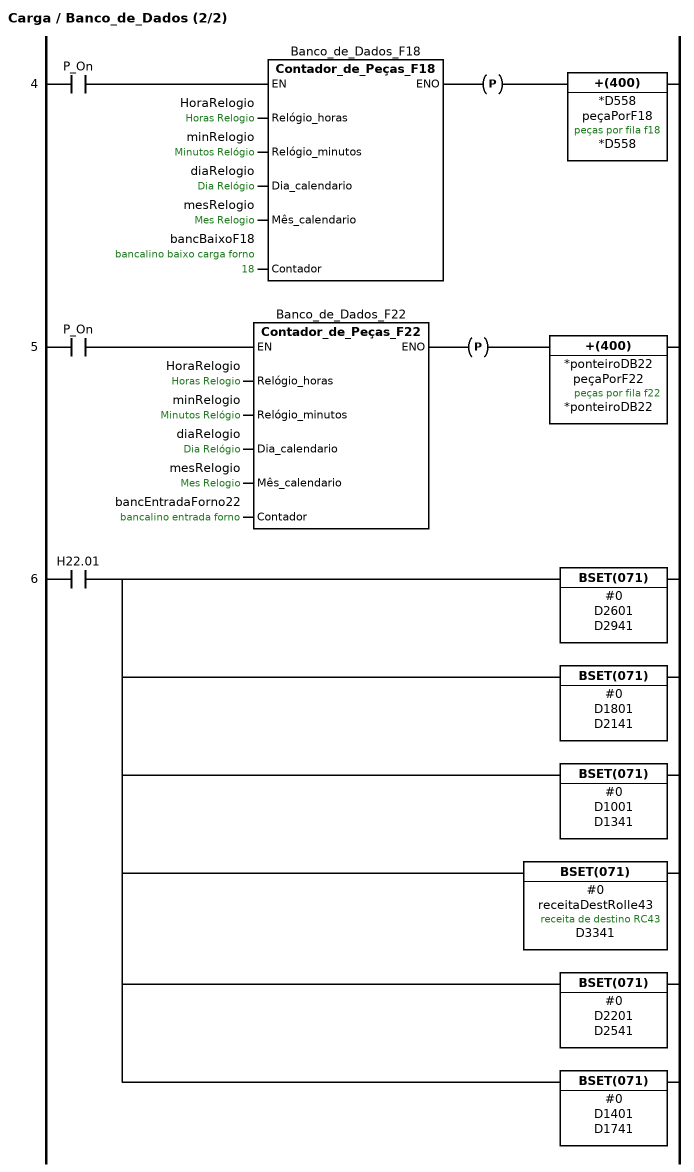
; [picture p24: Carga / Banco_de_Dados, rungs 4-6]
; rung 4
LD P_On
CALL Banco_de_Dados_F18 : Contador_de_Peças_F18 (Relógio_horas := HoraRelogio, Relógio_minutos := minRelogio, Dia_calendario := diaRelogio, Mês_calendario := mesRelogio, Contador := bancBaixoF18)  ; Horas Relogio, Minutos Relógio, Dia Relógio, Mes Relogio, bancalino baixo carga forno 18
UP(521)
+(400) *D558 peçaPorF18 *D558  ; peças por fila f18
; rung 5
LD P_On
CALL Banco_de_Dados_F22 : Contador_de_Peças_F22 (Relógio_horas := HoraRelogio, Relógio_minutos := minRelogio, Dia_calendario := diaRelogio, Mês_calendario := mesRelogio, Contador := bancEntradaForno22)  ; Horas Relogio, Minutos Relógio, Dia Relógio, Mes Relogio, bancalino entrada forno
UP(521)
+(400) *ponteiroDB22 peçaPorF22 *ponteiroDB22  ; peças por fila f22
; rung 6
LD H22.01
BSET(071) #0 D2601 D2941
BSET(071) #0 D1801 D2141
BSET(071) #0 D1001 D1341
BSET(071) #0 receitaDestRolle43 D3341  ; receita de destino RC43
BSET(071) #0 D2201 D2541
BSET(071) #0 D1401 D1741

### Section Transferencia_excel

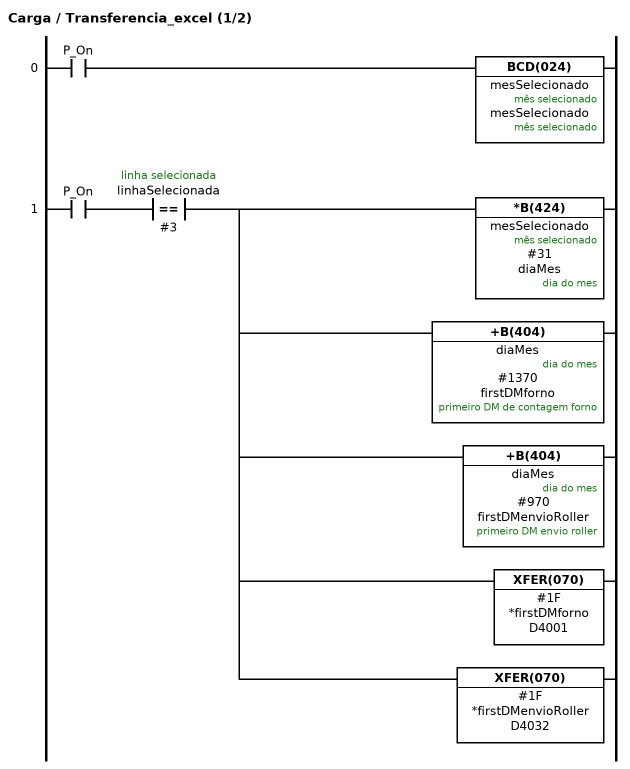
; rung 0
LD P_On
BCD(024) mesSelecionado mesSelecionado  ; mês selecionado
; rung 1
LD P_On
AND=(300) linhaSelecionada #3  ; linha selecionada
*B(424) mesSelecionado #31 diaMes  ; mês selecionado, dia do mes
+B(404) diaMes #1370 firstDMforno  ; dia do mes, primeiro DM de contagem forno
+B(404) diaMes #970 firstDMenvioRoller  ; dia do mes, primeiro DM envio roller
XFER(070) #1F *firstDMforno D4001
XFER(070) #1F *firstDMenvioRoller D4032

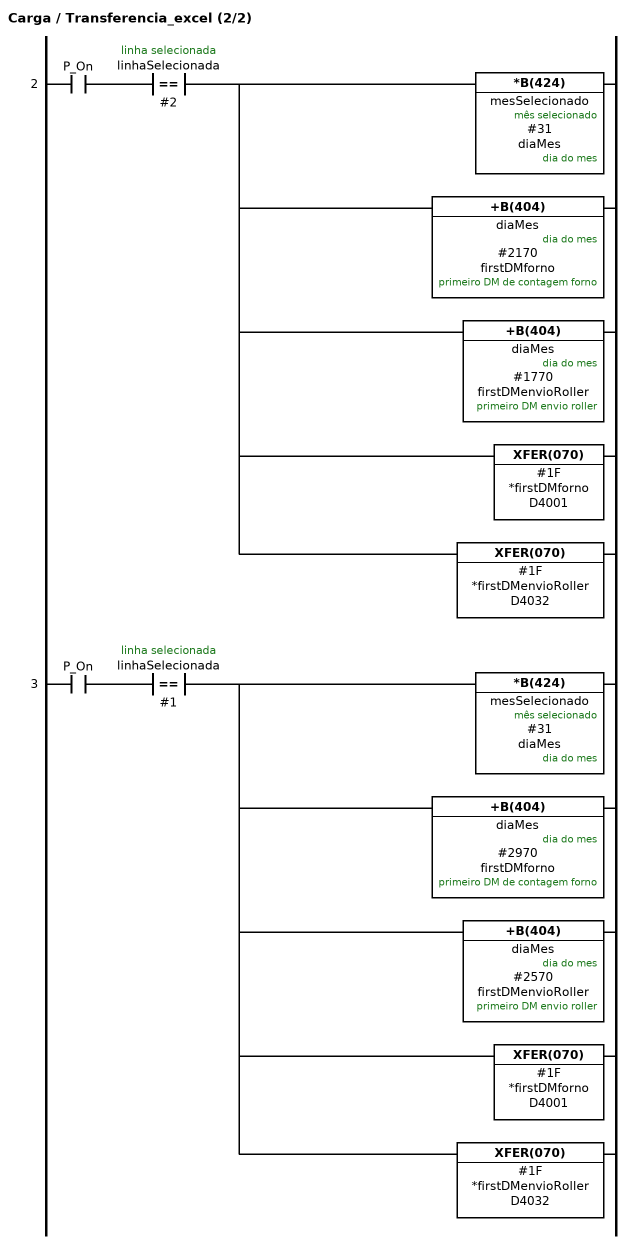
; rung 2
LD P_On
AND=(300) linhaSelecionada #2  ; linha selecionada
*B(424) mesSelecionado #31 diaMes  ; mês selecionado, dia do mes
+B(404) diaMes #2170 firstDMforno  ; dia do mes, primeiro DM de contagem forno
+B(404) diaMes #1770 firstDMenvioRoller  ; dia do mes, primeiro DM envio roller
XFER(070) #1F *firstDMforno D4001
XFER(070) #1F *firstDMenvioRoller D4032
; rung 3
LD P_On
AND=(300) linhaSelecionada #1  ; linha selecionada
*B(424) mesSelecionado #31 diaMes  ; mês selecionado, dia do mes
+B(404) diaMes #2970 firstDMforno  ; dia do mes, primeiro DM de contagem forno
+B(404) diaMes #2570 firstDMenvioRoller  ; dia do mes, primeiro DM envio roller
XFER(070) #1F *firstDMforno D4001
XFER(070) #1F *firstDMenvioRoller D4032

### Section Relogio

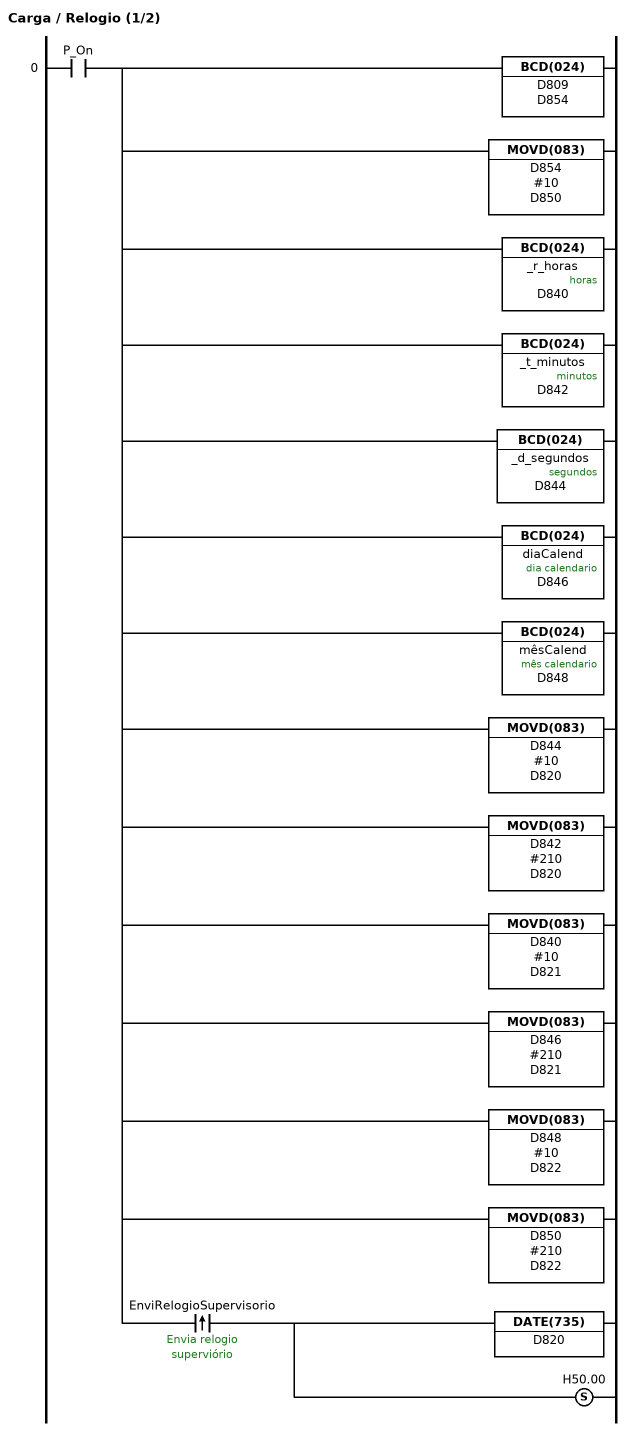
; rung 0
LD P_On
BCD(024) D809 D854
MOVD(083) D854 #10 D850
BCD(024) _r_horas D840  ; horas
BCD(024) _t_minutos D842  ; minutos
BCD(024) _d_segundos D844  ; segundos
BCD(024) diaCalend D846  ; dia calendario
BCD(024) mêsCalend D848  ; mês calendario
MOVD(083) D844 #10 D820
MOVD(083) D842 #210 D820
MOVD(083) D840 #10 D821
MOVD(083) D846 #210 D821
MOVD(083) D848 #10 D822
MOVD(083) D850 #210 D822
@AND EnviRelogioSupervisorio  ; Envia relogio superviório
DATE(735) D820
SET H50.00

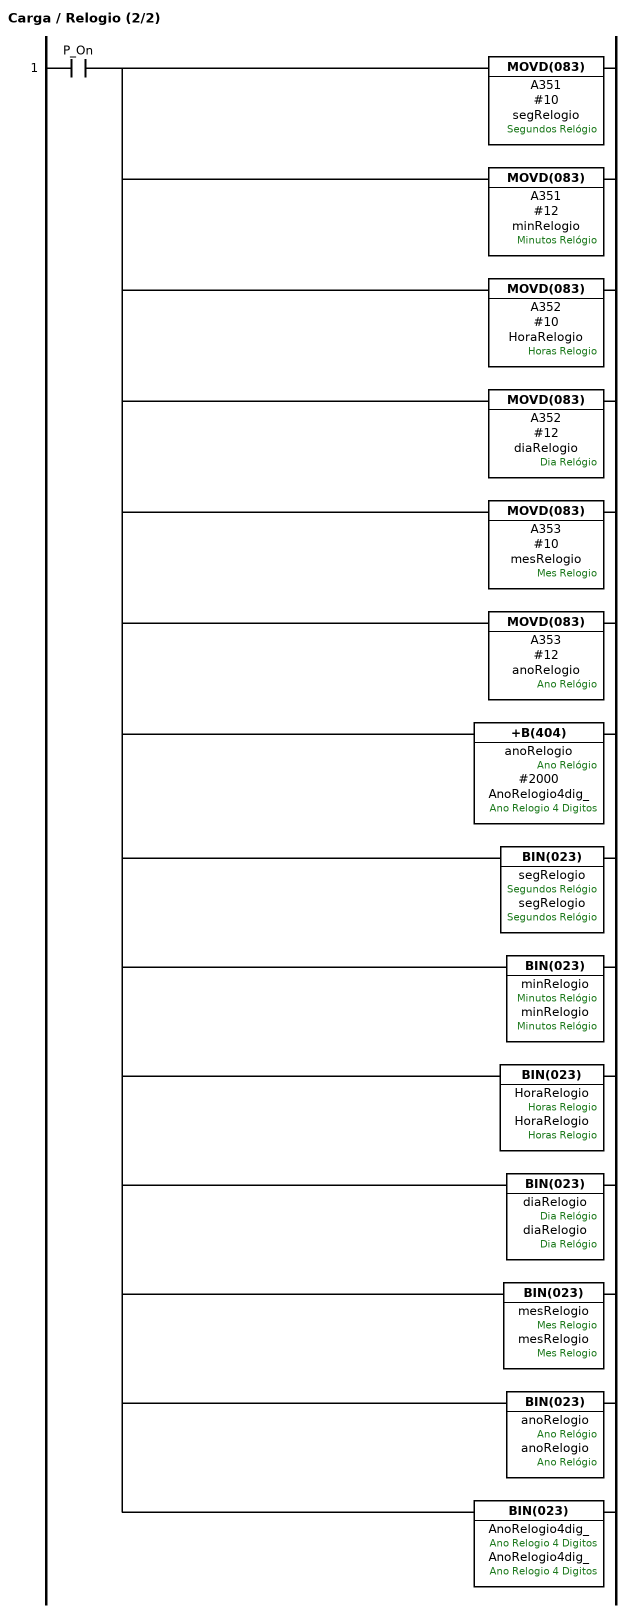
; rung 1
LD P_On
MOVD(083) A351 #10 segRelogio  ; Segundos Relógio
MOVD(083) A351 #12 minRelogio  ; Minutos Relógio
MOVD(083) A352 #10 HoraRelogio  ; Horas Relogio
MOVD(083) A352 #12 diaRelogio  ; Dia Relógio
MOVD(083) A353 #10 mesRelogio  ; Mes Relogio
MOVD(083) A353 #12 anoRelogio  ; Ano Relógio
+B(404) anoRelogio #2000 AnoRelogio4dig_  ; Ano Relógio, Ano Relogio 4 Digitos
BIN(023) segRelogio segRelogio  ; Segundos Relógio
BIN(023) minRelogio minRelogio  ; Minutos Relógio
BIN(023) HoraRelogio HoraRelogio  ; Horas Relogio
BIN(023) diaRelogio diaRelogio  ; Dia Relógio
BIN(023) mesRelogio mesRelogio  ; Mes Relogio
BIN(023) anoRelogio anoRelogio  ; Ano Relógio
BIN(023) AnoRelogio4dig_ AnoRelogio4dig_  ; Ano Relogio 4 Digitos

### Section End
; rung 0
END(001)

## Program Escolha41 (cyclic task 2)
Local symbols
TIM 4.12 BOOL
anoRelogio D328 CHANNEL  ; Ano relógio
bit2 BOOL
box1 4.01 BOOL  ; box1
box2 4.02 BOOL  ; box2
box3 4.03 BOOL  ; box3
box4 4.04 BOOL  ; box4
box5 4.05 BOOL  ; box5
box6 4.06 BOOL  ; box6
caco 4.00 BOOL  ; caco
cntAmostragem D316 CHANNEL  ; contador amostragem
cntBox0 D300 CHANNEL  ; contagem box 0
cntBox1 D302 CHANNEL  ; contagem box 1
cntBox2 D304 CHANNEL  ; contagem box 2
cntBox3 D306 CHANNEL  ; contagem box 3
cntBox4 D308 CHANNEL  ; contagem box 4
cntBox5 D310 CHANNEL  ; contagem box 5
cntBox6 D312 CHANNEL  ; contagem box 6
cntTotal D314 CHANNEL  ; contagem total
d400D400 CHANNEL
diaRelogio D324 CHANNEL  ; Dia relógio
enviaRelogio H12.00 BOOL  ; envia relogio
horEnvio D336 CHANNEL  ; hora de envio
horIHM D330 CHANNEL  ; hora ihm
horRelogio D322 CHANNEL  ; Horas relógio
mesRelogio D326 CHANNEL  ; Mes Relógio
minIHM D332 CHANNEL  ; minuto ihm
minRelogio D320 CHANNEL  ; Minutos relógio
mitEnvio D338 CHANNEL  ; minuto envio
resetCnt 4.07 BOOL  ; reset contagem
segEnvio D340 CHANNEL  ; segundo envio
segIHM D334 CHANNEL  ; segundo ihm
segRelogio D318 CHANNEL  ; Segundos Relógio
selecaoCom 4.09 BOOL  ; seleção comercial
totalPc 4.08 BOOL  ; total peças

### Section Controle_Qualidade

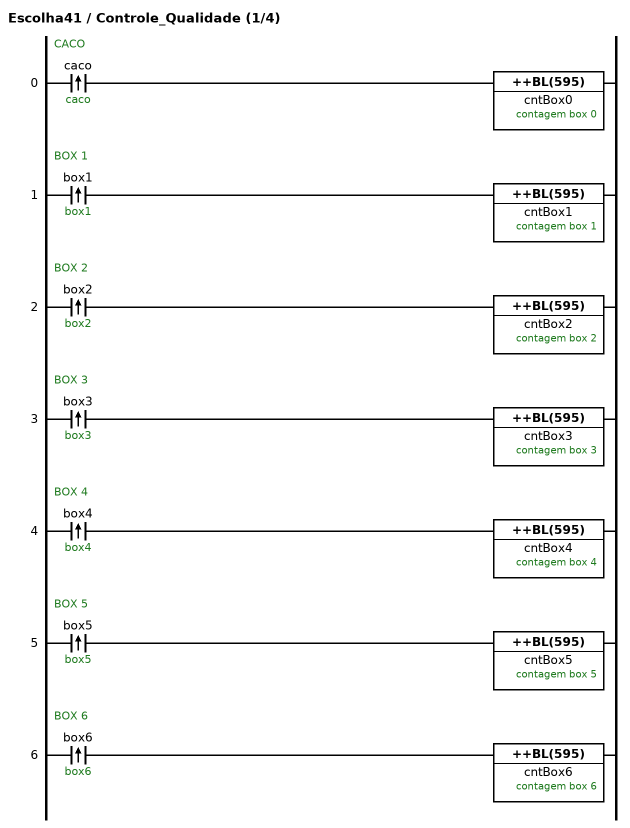
; rung 0: CACO
@LD caco  ; caco
++BL(595) cntBox0  ; contagem box 0
; rung 1: BOX 1
@LD box1  ; box1
++BL(595) cntBox1  ; contagem box 1
; rung 2: BOX 2
@LD box2  ; box2
++BL(595) cntBox2  ; contagem box 2
; rung 3: BOX 3
@LD box3  ; box3
++BL(595) cntBox3  ; contagem box 3
; rung 4: BOX 4
@LD box4  ; box4
++BL(595) cntBox4  ; contagem box 4
; rung 5: BOX 5
@LD box5  ; box5
++BL(595) cntBox5  ; contagem box 5
; rung 6: BOX 6
@LD box6  ; box6
++BL(595) cntBox6  ; contagem box 6

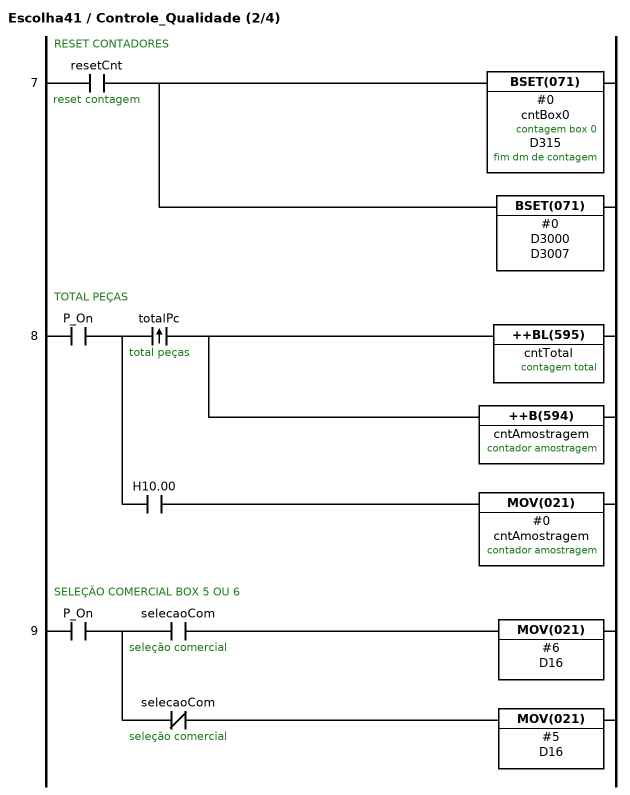
; rung 7: RESET CONTADORES
LD resetCnt  ; reset contagem
BSET(071) #0 cntBox0 D315  ; contagem box 0, fim dm de contagem
BSET(071) #0 D3000 D3007
; rung 8: TOTAL PEÇAS
LD P_On
OUT TR0
@AND totalPc  ; total peças
++BL(595) cntTotal  ; contagem total
++B(594) cntAmostragem  ; contador amostragem
LD TR0
AND H10.00
MOV(021) #0 cntAmostragem  ; contador amostragem
; rung 9: SELEÇÃO COMERCIAL BOX 5 OU 6
LD P_On
OUT TR0
AND selecaoCom  ; seleção comercial
MOV(021) #6 D16
LD TR0
ANDNOT selecaoCom  ; seleção comercial
MOV(021) #5 D16

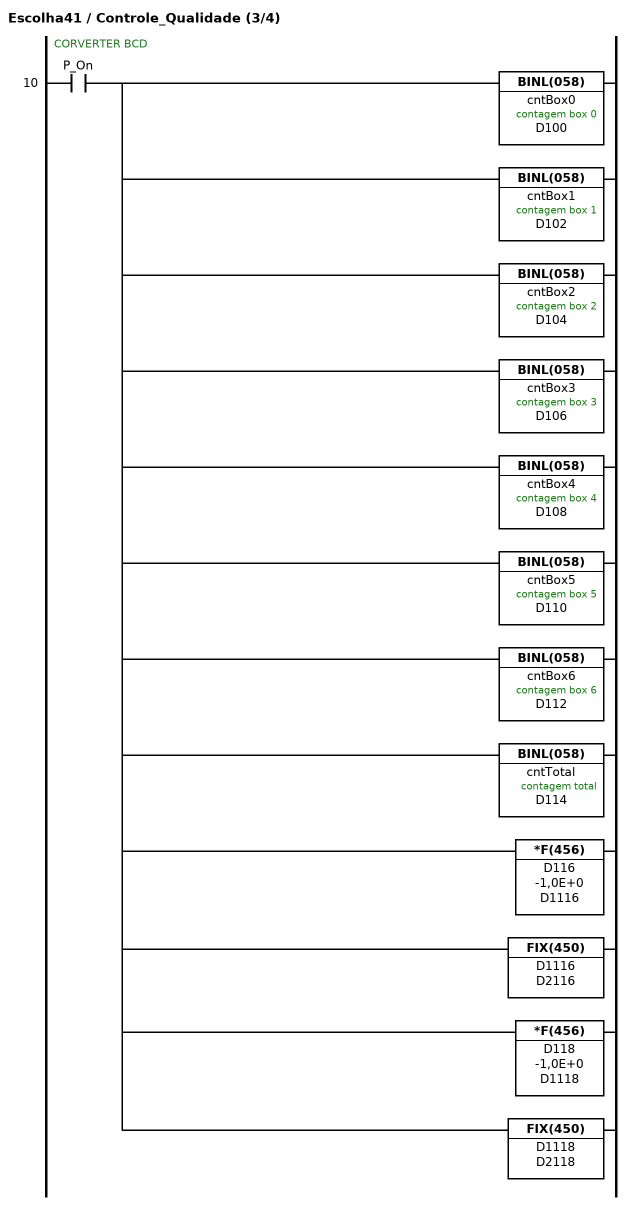
; rung 10: CORVERTER BCD
LD P_On
BINL(058) cntBox0 D100  ; contagem box 0
BINL(058) cntBox1 D102  ; contagem box 1
BINL(058) cntBox2 D104  ; contagem box 2
BINL(058) cntBox3 D106  ; contagem box 3
BINL(058) cntBox4 D108  ; contagem box 4
BINL(058) cntBox5 D110  ; contagem box 5
BINL(058) cntBox6 D112  ; contagem box 6
BINL(058) cntTotal D114  ; contagem total
*F(456) D116 -1,0E+0 D1116
FIX(450) D1116 D2116
*F(456) D118 -1,0E+0 D1118
FIX(450) D1118 D2118

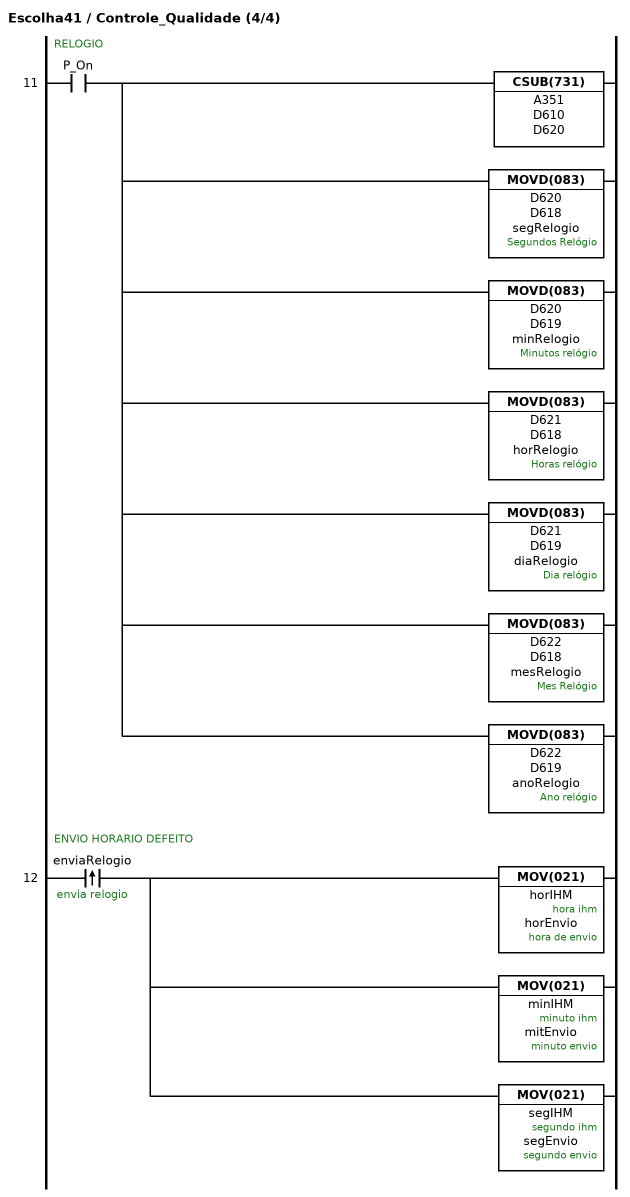
; rung 11: RELOGIO
LD P_On
CSUB(731) A351 D610 D620
MOVD(083) D620 D618 segRelogio  ; Segundos Relógio
MOVD(083) D620 D619 minRelogio  ; Minutos relógio
MOVD(083) D621 D618 horRelogio  ; Horas relógio
MOVD(083) D621 D619 diaRelogio  ; Dia relógio
MOVD(083) D622 D618 mesRelogio  ; Mes Relógio
MOVD(083) D622 D619 anoRelogio  ; Ano relógio
; rung 12: ENVIO HORARIO DEFEITO
@LD enviaRelogio  ; envia relogio
MOV(021) horIHM horEnvio  ; hora ihm, hora de envio
MOV(021) minIHM mitEnvio  ; minuto ihm, minuto envio
MOV(021) segIHM segEnvio  ; segundo ihm, segundo envio

### Section END
; rung 0
END(001)

## Program Escolha43 (cyclic task 3)
Local symbols
TIM 5.12 BOOL
anoRelogio D428 CHANNEL  ; Ano relógio
bit2 BOOL
box1 5.01 BOOL  ; box1
box2 5.02 BOOL  ; box2
box3 5.03 BOOL  ; box3
box4 5.04 BOOL  ; box4
box5 5.05 BOOL  ; box5
box6 5.06 BOOL  ; box6
caco 5.00 BOOL  ; caco
cntAmostragem D416 CHANNEL  ; contador amostragem
cntBox0 D400 CHANNEL  ; contagem box 0
cntBox1 D402 CHANNEL  ; contagem box 1
cntBox2 D404 CHANNEL  ; contagem box 2
cntBox3 D406 CHANNEL  ; contagem box 3
cntBox4 D408 CHANNEL  ; contagem box 4
cntBox5 D410 CHANNEL  ; contagem box 5
cntBox6 D412 CHANNEL  ; contagem box 6
cntTotal D414 CHANNEL  ; contagem total
d400D400 CHANNEL
diaRelogio D424 CHANNEL  ; Dia relógio
enviaRelogio H13.01 BOOL  ; envia relogio
horEnvio D436 CHANNEL  ; hora de envio
horIHM D430 CHANNEL  ; hora ihm
horRelogio D422 CHANNEL  ; Horas relógio
mesRelogio D426 CHANNEL  ; Mes Relógio
minIHM D432 CHANNEL  ; minuto ihm
minRelogio D420 CHANNEL  ; Minutos relógio
mitEnvio D438 CHANNEL  ; minuto envio
resetCnt 5.07 BOOL  ; reset contagem
resetCntH H13.00 BOOL  ; reset contador
segEnvio D440 CHANNEL  ; segundo envio
segIHM D434 CHANNEL  ; segundo ihm
segRelogio D418 CHANNEL  ; Segundos Relógio
selecaoCom 5.09 BOOL  ; seleção comercial
totalPc 5.08 BOOL  ; total peças

### Section Controle_Qualidade

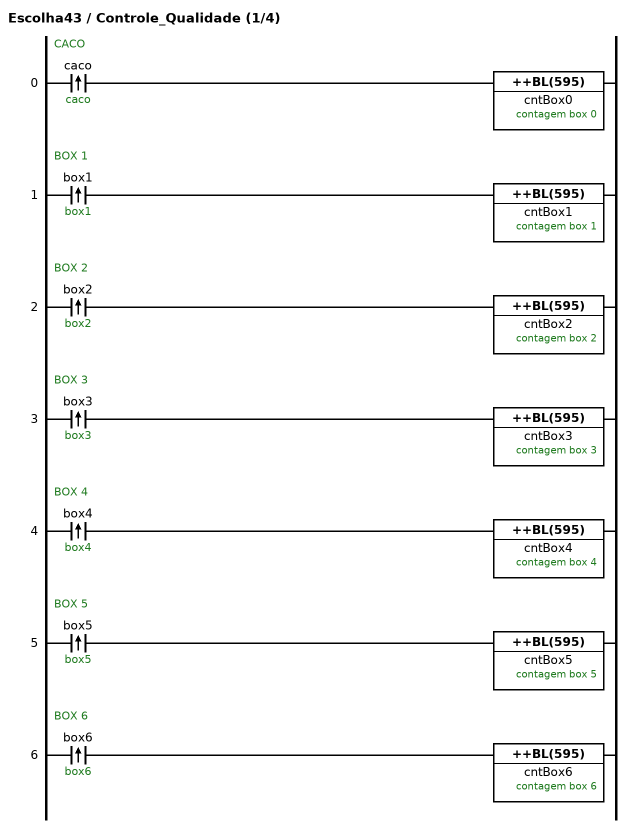
; rung 0: CACO
@LD caco  ; caco
++BL(595) cntBox0  ; contagem box 0
; rung 1: BOX 1
@LD box1  ; box1
++BL(595) cntBox1  ; contagem box 1
; rung 2: BOX 2
@LD box2  ; box2
++BL(595) cntBox2  ; contagem box 2
; rung 3: BOX 3
@LD box3  ; box3
++BL(595) cntBox3  ; contagem box 3
; rung 4: BOX 4
@LD box4  ; box4
++BL(595) cntBox4  ; contagem box 4
; rung 5: BOX 5
@LD box5  ; box5
++BL(595) cntBox5  ; contagem box 5
; rung 6: BOX 6
@LD box6  ; box6
++BL(595) cntBox6  ; contagem box 6

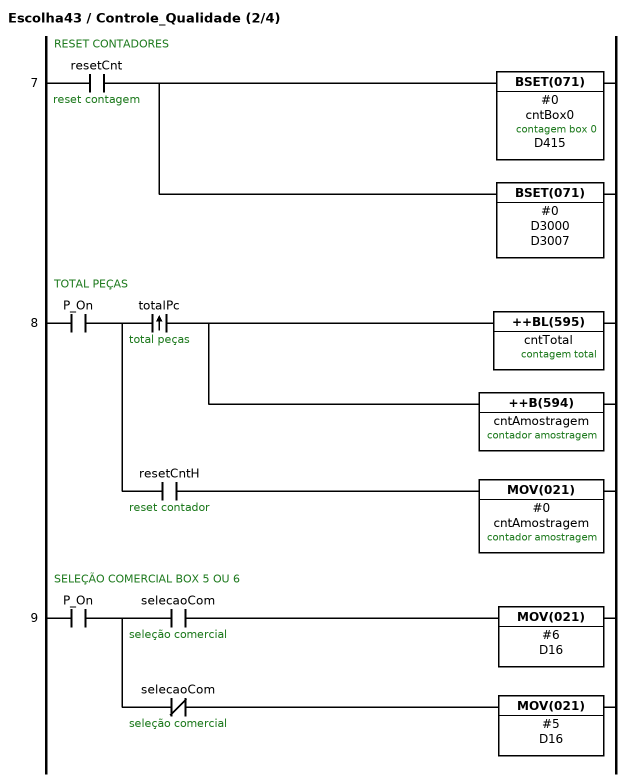
; rung 7: RESET CONTADORES
LD resetCnt  ; reset contagem
BSET(071) #0 cntBox0 D415  ; contagem box 0
BSET(071) #0 D3000 D3007
; rung 8: TOTAL PEÇAS
LD P_On
OUT TR0
@AND totalPc  ; total peças
++BL(595) cntTotal  ; contagem total
++B(594) cntAmostragem  ; contador amostragem
LD TR0
AND resetCntH  ; reset contador
MOV(021) #0 cntAmostragem  ; contador amostragem
; rung 9: SELEÇÃO COMERCIAL BOX 5 OU 6
LD P_On
OUT TR0
AND selecaoCom  ; seleção comercial
MOV(021) #6 D16
LD TR0
ANDNOT selecaoCom  ; seleção comercial
MOV(021) #5 D16

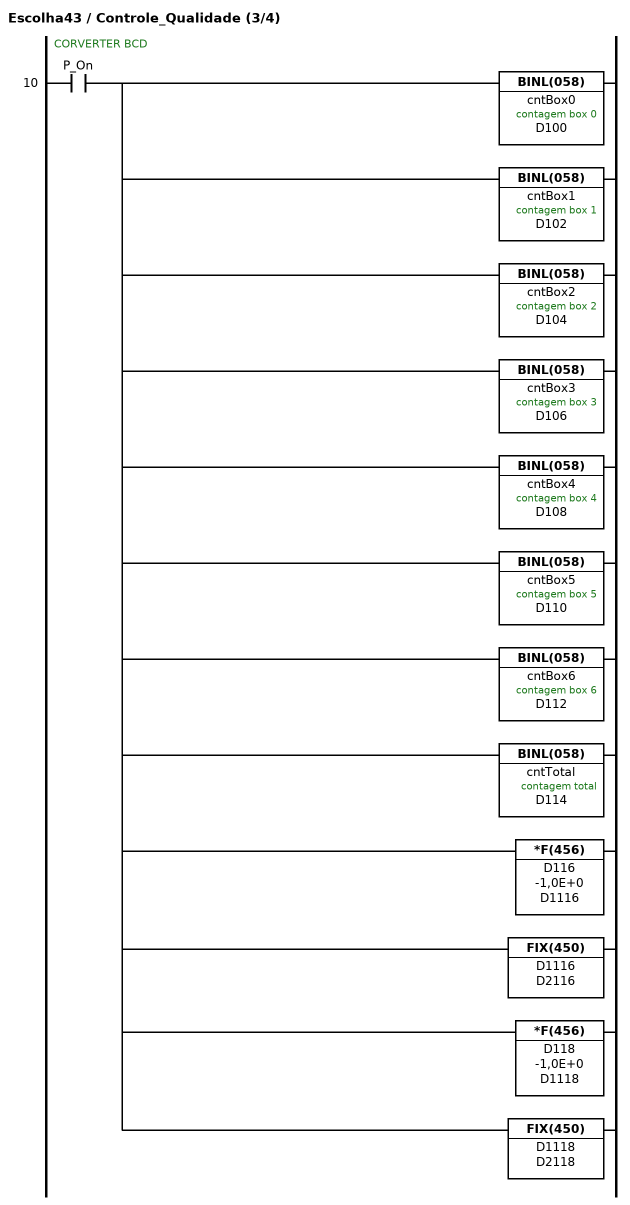
; rung 10: CORVERTER BCD
LD P_On
BINL(058) cntBox0 D100  ; contagem box 0
BINL(058) cntBox1 D102  ; contagem box 1
BINL(058) cntBox2 D104  ; contagem box 2
BINL(058) cntBox3 D106  ; contagem box 3
BINL(058) cntBox4 D108  ; contagem box 4
BINL(058) cntBox5 D110  ; contagem box 5
BINL(058) cntBox6 D112  ; contagem box 6
BINL(058) cntTotal D114  ; contagem total
*F(456) D116 -1,0E+0 D1116
FIX(450) D1116 D2116
*F(456) D118 -1,0E+0 D1118
FIX(450) D1118 D2118

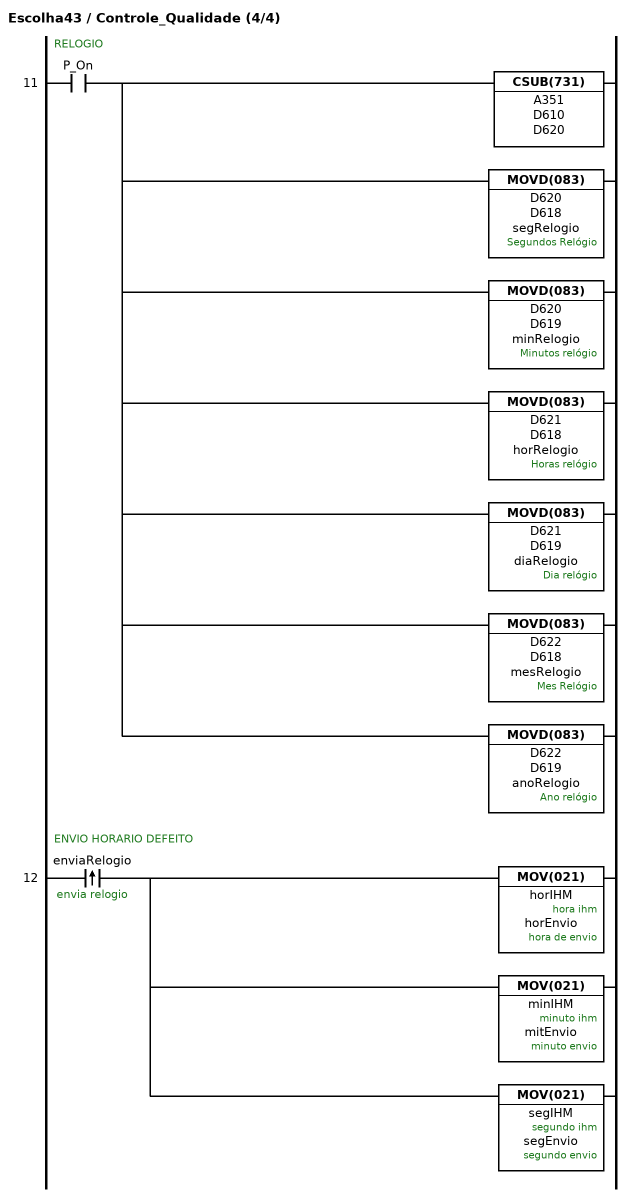
; rung 11: RELOGIO
LD P_On
CSUB(731) A351 D610 D620
MOVD(083) D620 D618 segRelogio  ; Segundos Relógio
MOVD(083) D620 D619 minRelogio  ; Minutos relógio
MOVD(083) D621 D618 horRelogio  ; Horas relógio
MOVD(083) D621 D619 diaRelogio  ; Dia relógio
MOVD(083) D622 D618 mesRelogio  ; Mes Relógio
MOVD(083) D622 D619 anoRelogio  ; Ano relógio
; rung 12: ENVIO HORARIO DEFEITO
@LD enviaRelogio  ; envia relogio
MOV(021) horIHM horEnvio  ; hora ihm, hora de envio
MOV(021) minIHM mitEnvio  ; minuto ihm, minuto envio
MOV(021) segIHM segEnvio  ; segundo ihm, segundo envio

### Section END
; rung 0
END(001)

## Function block Contador_de_Peças_F17
VAR_INPUT
  Relógio_horas : WORD;
  Relógio_minutos : WORD;
  Dia_calendario : WORD;
  Mês_calendario : WORD;
  Contador : BOOL;
END_VAR
VAR
  _31dias_vezes_2 AT D530 : WORD;
  Ponteiro_DWord AT D532 : WORD;
  Memória_de_Armazenagem AT D534 : WORD;
  Memoria_contagem_BIN AT D536 : WORD;
  Memoria_contagem_BCD AT D538 : WORD;
END_VAR

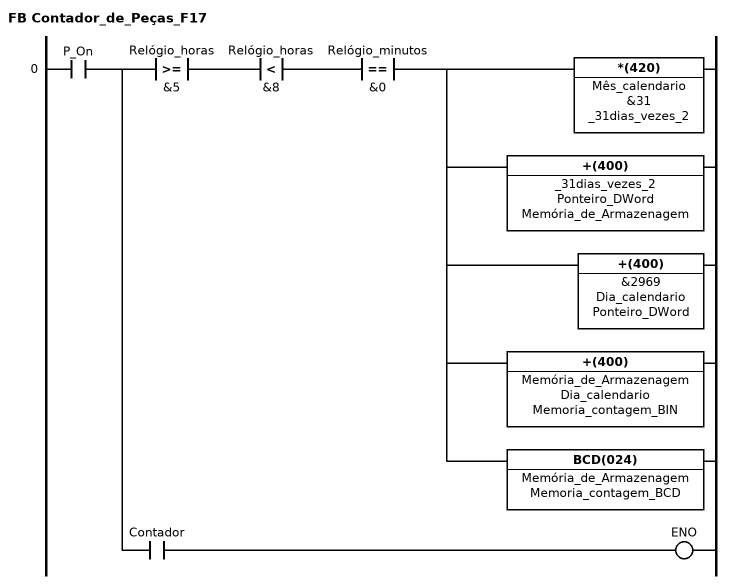
; rung 0
LD P_On
OUT TR0
AND>=(325) Relógio_horas &5
AND<(310) Relógio_horas &8
AND=(300) Relógio_minutos &0
*(420) Mês_calendario &31 _31dias_vezes_2
+(400) _31dias_vezes_2 Ponteiro_DWord Memória_de_Armazenagem
+(400) &2969 Dia_calendario Ponteiro_DWord
+(400) Memória_de_Armazenagem Dia_calendario Memoria_contagem_BIN
BCD(024) Memória_de_Armazenagem Memoria_contagem_BCD
LD TR0
AND Contador
OUT ENO

## Function block Contador_de_Peças_F18
VAR_INPUT
  Relógio_horas : WORD;
  Relógio_minutos : WORD;
  Dia_calendario : WORD;
  Mês_calendario : WORD;
  Contador : BOOL;
END_VAR
VAR
  _31dias_vezes_2 AT D550 : WORD;
  Ponteiro_DWord AT D552 : WORD;
  Memória_de_Armazenagem AT D554 : WORD;
  Memoria_contagem_BIN AT D556 : WORD;
  Memoria_contagem_BCD AT D558 : WORD;
END_VAR

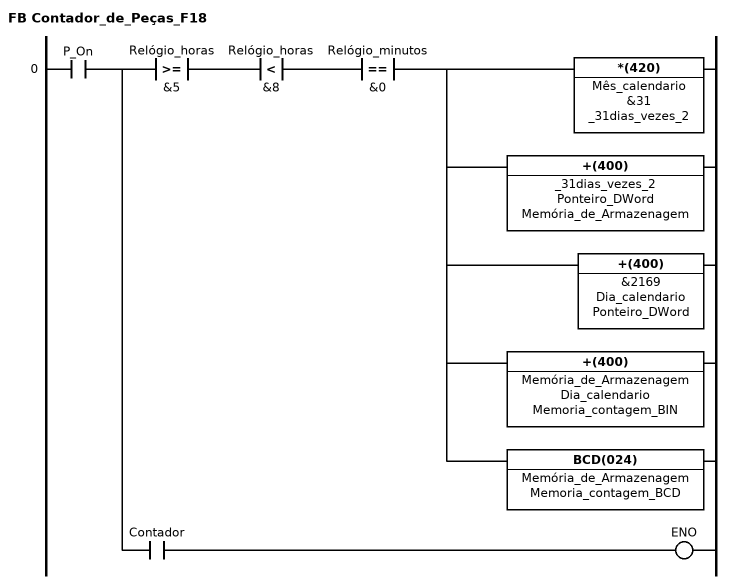
; rung 0
LD P_On
OUT TR0
AND>=(325) Relógio_horas &5
AND<(310) Relógio_horas &8
AND=(300) Relógio_minutos &0
*(420) Mês_calendario &31 _31dias_vezes_2
+(400) _31dias_vezes_2 Ponteiro_DWord Memória_de_Armazenagem
+(400) &2169 Dia_calendario Ponteiro_DWord
+(400) Memória_de_Armazenagem Dia_calendario Memoria_contagem_BIN
BCD(024) Memória_de_Armazenagem Memoria_contagem_BCD
LD TR0
AND Contador
OUT ENO

## Function block Contador_de_Peças_F22
VAR_INPUT
  Relógio_horas : WORD;
  Relógio_minutos : WORD;
  Dia_calendario : WORD;
  Mês_calendario : WORD;
  Contador : BOOL;
END_VAR
VAR
  _31dias_vezes_2 AT D510 : WORD;
  Ponteiro_DWord AT D512 : WORD;
  Memória_de_Armazenagem AT D514 : WORD;
  Memoria_contagem_BIN AT D516 : WORD;
  Memoria_contagem_BCD AT D518 : WORD;
END_VAR

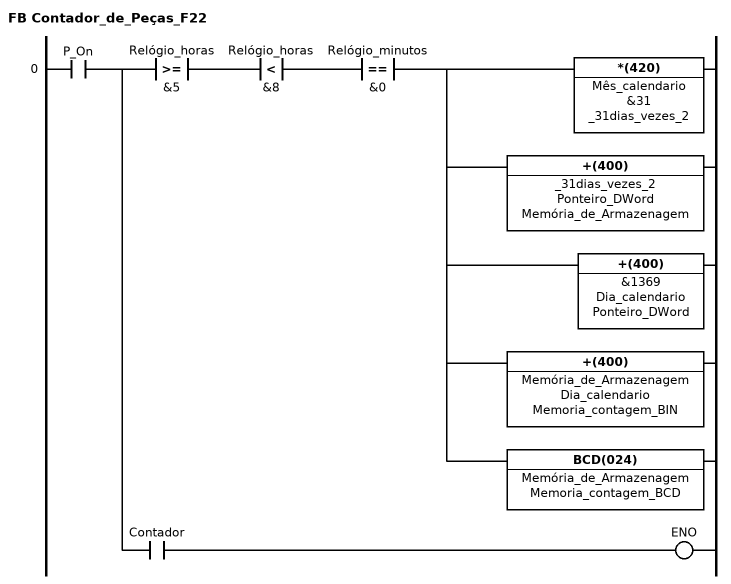
; rung 0
LD P_On
OUT TR0
AND>=(325) Relógio_horas &5
AND<(310) Relógio_horas &8
AND=(300) Relógio_minutos &0
*(420) Mês_calendario &31 _31dias_vezes_2
+(400) _31dias_vezes_2 Ponteiro_DWord Memória_de_Armazenagem
+(400) &1369 Dia_calendario Ponteiro_DWord
+(400) Memória_de_Armazenagem Dia_calendario Memoria_contagem_BIN
BCD(024) Memória_de_Armazenagem Memoria_contagem_BCD
LD TR0
AND Contador
OUT ENO

## Function block Contador_de_Peças_PH29
VAR_INPUT
  Relógio_horas : WORD;
  Relógio_minutos : WORD;
  Dia_calendario : WORD;
  Mês_calendario : WORD;
  Contador : BOOL;
END_VAR
VAR
  _31dias_vezes_2 AT D520 : WORD;
  Ponteiro_DWord AT D522 : WORD;
  Memória_de_Armazenagem AT D524 : WORD;
  Memoria_contagem_BIN AT D526 : WORD;
  Memoria_contagem_BCD AT D528 : WORD;
END_VAR

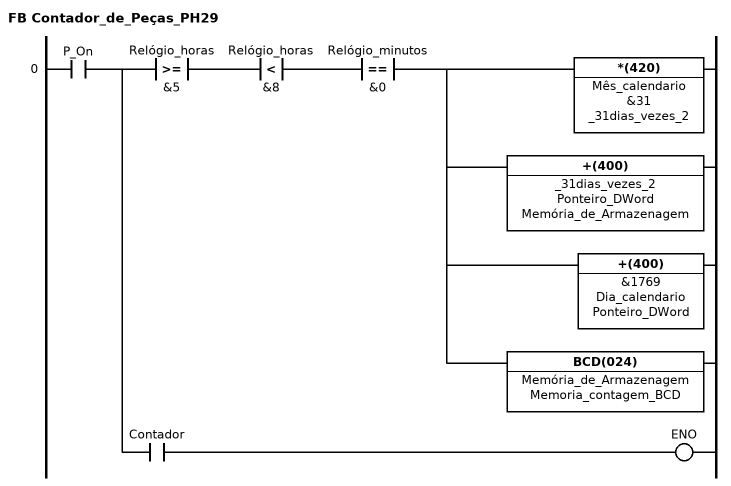
; rung 0
LD P_On
OUT TR0
AND>=(325) Relógio_horas &5
AND<(310) Relógio_horas &8
AND=(300) Relógio_minutos &0
*(420) Mês_calendario &31 _31dias_vezes_2
+(400) _31dias_vezes_2 Ponteiro_DWord Memória_de_Armazenagem
+(400) &1769 Dia_calendario Ponteiro_DWord
BCD(024) Memória_de_Armazenagem Memoria_contagem_BCD
LD TR0
AND Contador
OUT ENO

## Function block Contador_de_Peças_PH30
VAR_INPUT
  Relógio_horas : WORD;
  Relógio_minutos : WORD;
  Dia_calendario : WORD;
  Mês_calendario : WORD;
  Contador : BOOL;
END_VAR
VAR
  _31dias_vezes_2 AT D510 : WORD;
  Ponteiro_DWord AT D512 : WORD;
  Memória_de_Armazenagem AT D514 : WORD;
  Memoria_contagem_BIN AT D516 : WORD;
  Memoria_contagem_BCD AT D518 : WORD;
END_VAR

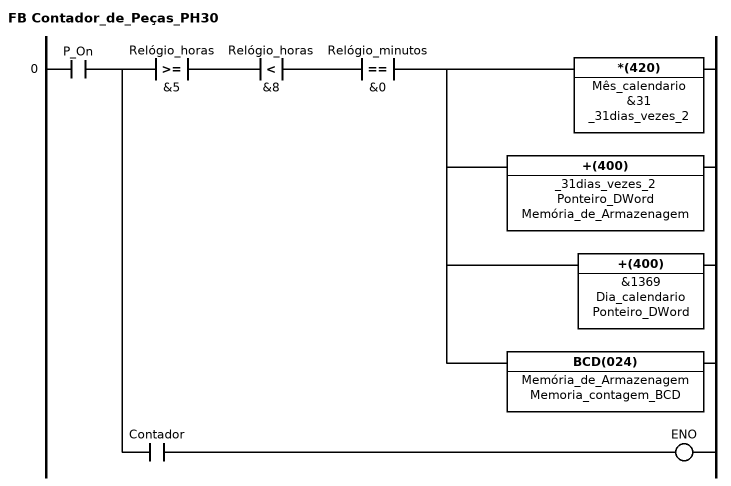
; rung 0
LD P_On
OUT TR0
AND>=(325) Relógio_horas &5
AND<(310) Relógio_horas &8
AND=(300) Relógio_minutos &0
*(420) Mês_calendario &31 _31dias_vezes_2
+(400) _31dias_vezes_2 Ponteiro_DWord Memória_de_Armazenagem
+(400) &1369 Dia_calendario Ponteiro_DWord
BCD(024) Memória_de_Armazenagem Memoria_contagem_BCD
LD TR0
AND Contador
OUT ENO

## Function block Contador_de_Peças_PH31
VAR_INPUT
  Relógio_horas : WORD;
  Relógio_minutos : WORD;
  Dia_calendario : WORD;
  Mês_calendario : WORD;
  Contador : BOOL;
END_VAR
VAR
  _31dias_vezes_2 AT D500 : WORD;
  Ponteiro_DWord AT D502 : WORD;
  Memória_de_Armazenagem AT D504 : WORD;
  Memoria_contagem_BIN AT D506 : WORD;
  Memoria_contagem_BCD AT D508 : WORD;
END_VAR

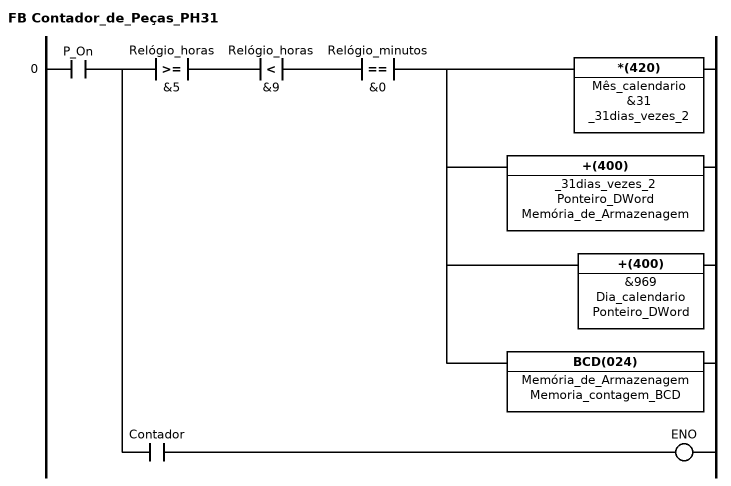
; rung 0
LD P_On
OUT TR0
AND>=(325) Relógio_horas &5
AND<(310) Relógio_horas &9
AND=(300) Relógio_minutos &0
*(420) Mês_calendario &31 _31dias_vezes_2
+(400) _31dias_vezes_2 Ponteiro_DWord Memória_de_Armazenagem
+(400) &969 Dia_calendario Ponteiro_DWord
BCD(024) Memória_de_Armazenagem Memoria_contagem_BCD
LD TR0
AND Contador
OUT ENO

## Function block Contador_de_Peças_RC41
VAR_INPUT
  Relógio_horas : WORD;
  Relógio_minutos : WORD;
  Dia_calendario : WORD;
  Mês_calendario : WORD;
  Contador : BOOL;
END_VAR
VAR
  _31dias_vezes_2 AT D520 : WORD;
  Ponteiro_DWord AT D522 : WORD;
  Memória_de_Armazenagem AT D524 : WORD;
  Memoria_contagem_BIN AT D526 : WORD;
  Memoria_contagem_BCD AT D528 : WORD;
END_VAR

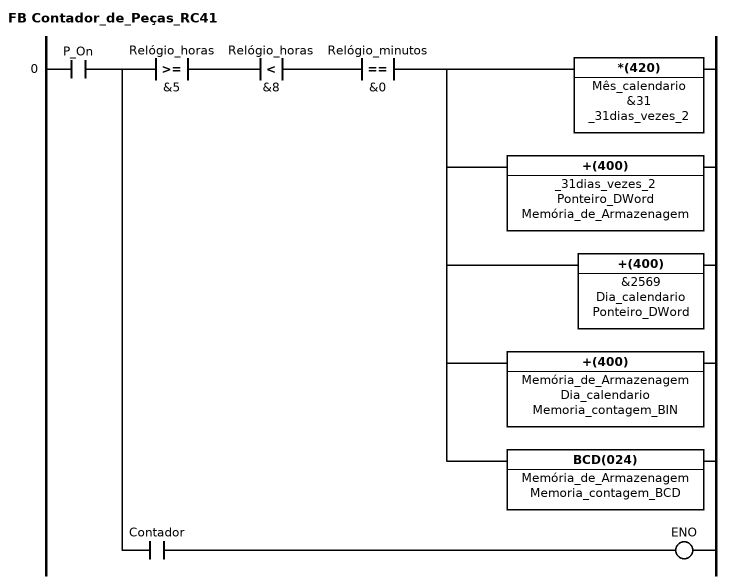
; rung 0
LD P_On
OUT TR0
AND>=(325) Relógio_horas &5
AND<(310) Relógio_horas &8
AND=(300) Relógio_minutos &0
*(420) Mês_calendario &31 _31dias_vezes_2
+(400) _31dias_vezes_2 Ponteiro_DWord Memória_de_Armazenagem
+(400) &2569 Dia_calendario Ponteiro_DWord
+(400) Memória_de_Armazenagem Dia_calendario Memoria_contagem_BIN
BCD(024) Memória_de_Armazenagem Memoria_contagem_BCD
LD TR0
AND Contador
OUT ENO

## Function block Contador_de_Peças_RC42
VAR_INPUT
  Relógio_horas : WORD;
  Relógio_minutos : WORD;
  Dia_calendario : WORD;
  Mês_calendario : WORD;
  Contador : BOOL;
END_VAR
VAR
  _31dias_vezes_2 AT D540 : WORD;
  Ponteiro_DWord AT D542 : WORD;
  Memória_de_Armazenagem AT D544 : WORD;
  Memoria_contagem_BIN AT D546 : WORD;
  Memoria_contagem_BCD AT D548 : WORD;
END_VAR

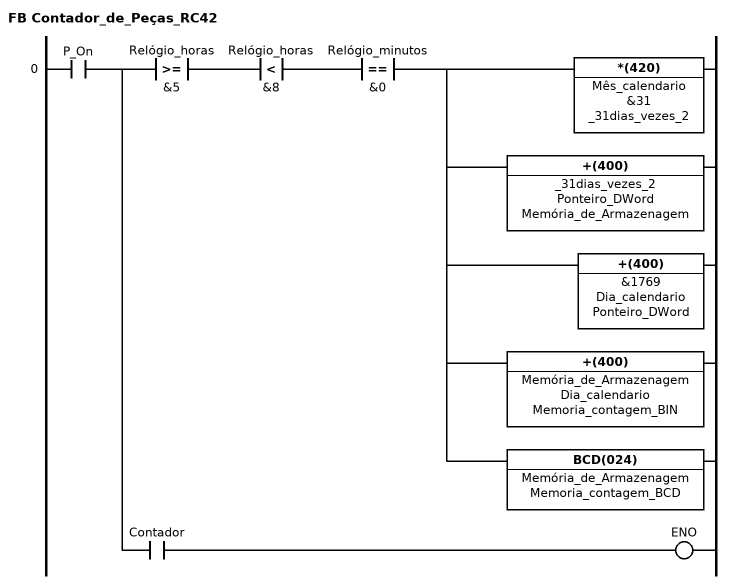
; rung 0
LD P_On
OUT TR0
AND>=(325) Relógio_horas &5
AND<(310) Relógio_horas &8
AND=(300) Relógio_minutos &0
*(420) Mês_calendario &31 _31dias_vezes_2
+(400) _31dias_vezes_2 Ponteiro_DWord Memória_de_Armazenagem
+(400) &1769 Dia_calendario Ponteiro_DWord
+(400) Memória_de_Armazenagem Dia_calendario Memoria_contagem_BIN
BCD(024) Memória_de_Armazenagem Memoria_contagem_BCD
LD TR0
AND Contador
OUT ENO

## Function block Contador_de_Peças_RC43
VAR_INPUT
  Relógio_horas : WORD;
  Relógio_minutos : WORD;
  Dia_calendario : WORD;
  Mês_calendario : WORD;
  Contador : BOOL;
END_VAR
VAR
  _31dias_vezes_2 AT D500 : WORD;
  Ponteiro_DWord AT D502 : WORD;
  Memória_de_Armazenagem AT D504 : WORD;
  Memoria_contagem_BIN AT D506 : WORD;
  Memoria_contagem_BCD AT D508 : WORD;
END_VAR

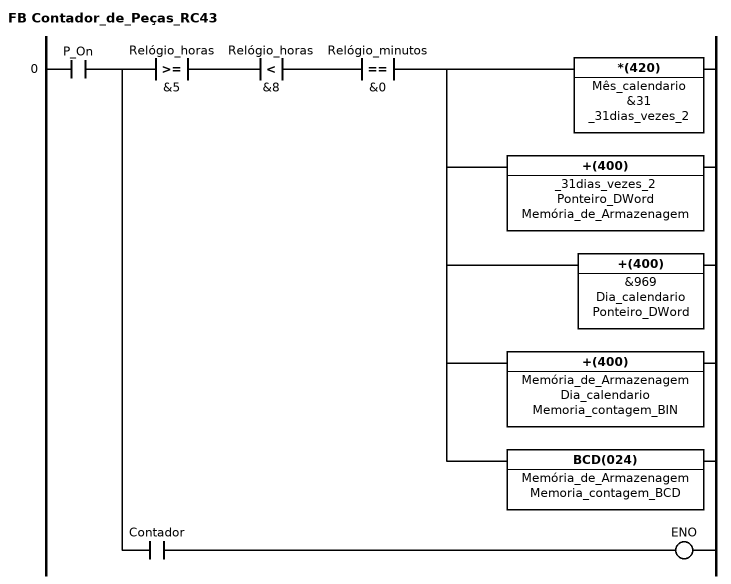
; rung 0
LD P_On
OUT TR0
AND>=(325) Relógio_horas &5
AND<(310) Relógio_horas &8
AND=(300) Relógio_minutos &0
*(420) Mês_calendario &31 _31dias_vezes_2
+(400) _31dias_vezes_2 Ponteiro_DWord Memória_de_Armazenagem
+(400) &969 Dia_calendario Ponteiro_DWord
+(400) Memória_de_Armazenagem Dia_calendario Memoria_contagem_BIN
BCD(024) Memória_de_Armazenagem Memoria_contagem_BCD
LD TR0
AND Contador
OUT ENO

## Function block Formato_de_Trabalho_29
VAR_INPUT
  Dia_calendario : WORD;
  Mês_calendario : WORD;
END_VAR
VAR
  _31dias_vezes_2 AT D546 : WORD;
  Ponteiro_DWord AT D548 : WORD;
  Memória_de_Armazenagem AT D550 : WORD;
  Memoria_contagem_BCD AT D552 : WORD;
END_VAR

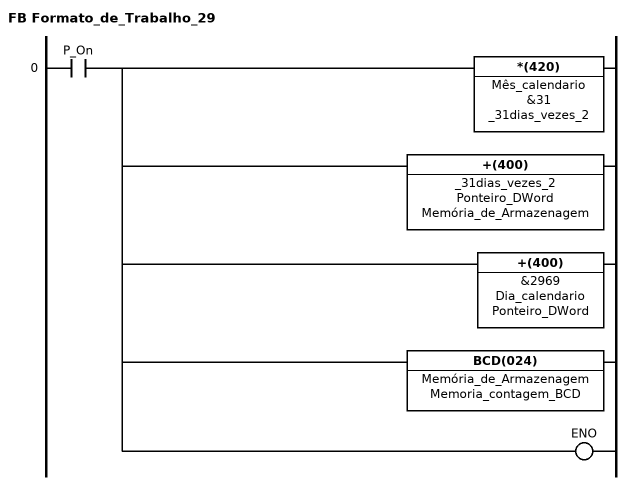
; rung 0
LD P_On
*(420) Mês_calendario &31 _31dias_vezes_2
+(400) _31dias_vezes_2 Ponteiro_DWord Memória_de_Armazenagem
+(400) &2969 Dia_calendario Ponteiro_DWord
BCD(024) Memória_de_Armazenagem Memoria_contagem_BCD
OUT ENO

## Function block Formato_de_Trabalho_30
VAR_INPUT
  Dia_calendario : WORD;
  Mês_calendario : WORD;
END_VAR
VAR
  _31dias_vezes_2 AT D538 : WORD;
  Ponteiro_DWord AT D540 : WORD;
  Memória_de_Armazenagem AT D542 : WORD;
  Memoria_contagem_BCD AT D544 : WORD;
END_VAR

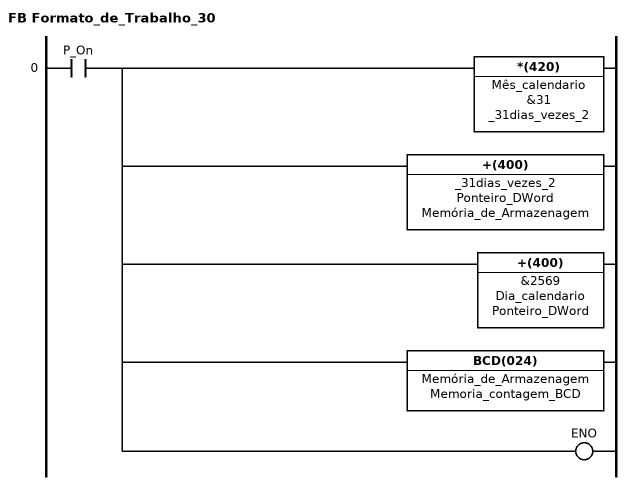
; rung 0
LD P_On
*(420) Mês_calendario &31 _31dias_vezes_2
+(400) _31dias_vezes_2 Ponteiro_DWord Memória_de_Armazenagem
+(400) &2569 Dia_calendario Ponteiro_DWord
BCD(024) Memória_de_Armazenagem Memoria_contagem_BCD
OUT ENO

## Function block Formato_de_Trabalho_31
VAR_INPUT
  Dia_calendario : WORD;
  Mês_calendario : WORD;
END_VAR
VAR
  _31dias_vezes_2 AT D530 : WORD;
  Ponteiro_DWord AT D532 : WORD;
  Memória_de_Armazenagem AT D534 : WORD;
  Memoria_contagem_BCD AT D536 : WORD;
END_VAR

